Staubli VAL3: Day14.dtx

string sInput
lists lResult
  [0]
    string sString
num nResult
string sStart
string sCombo[2]
string sResult
string sUnique
lists lSplit
  [0]
    string sString
lists_string_num lStrNum
  [0]
    string sString
    num nNum
num nUnique
